FUNCTION_BLOCK FB_AdsLog
VAR_INPUT
END_VAR
VAR_OUTPUT
END_VAR
VAR
	reBtnReset	: R_TRIG;						// Flankenerkennng für Meldeauslösung
	udiAdsLogResStr	: DINT;						// Aufrufergebnis 0 = i.O. oder Fehlercode
	strMessageVariable	: STRING := 'Reset';	// Variabler Meldetext
	
END_VAR


reBtnReset(CLK:=GVL_C1.S01_C1_SF16);
IF reBtnReset.Q THEN
	udiAdsLogResStr:= ADSLOGSTR(msgCtrlMask:=	ADSLOG_MSGTYPE_WARN 
												OR ADSLOG_MSGTYPE_LOG 
												OR ADSLOG_MSGTYPE_MSGBOX ,
												 msgFmtStr:= 'Betätigte Taste: %s',
												strArg:=strMessageVariable );
END_IF;

END_FUNCTION_BLOCK

(* stored: Version 1.1.0.1, ProductVersion 3.1.4024.12
   POU FB_AdsLog: Id {a5c9d88e-2503-4d87-ba56-4ab86a7d3854}, SpecialFunc None *)
